PROGRAM MAIN
VAR
	Axis1 : AXIS_REF;
	
	PowerAxis1 : MC_Power;
	PowerAxis1Out : ST_McOutputs;
	
	ResetAxis1 : MC_Reset;
	ResetAxis1Out : ST_McOutputs;
	
	MoveAxis1 : MC_MoveAbsolute();
	MoveAxis2 : MC_MoveAbsolute;
	MoveAbsolute1 : ST_McOutputs;
	MoveAbsolute2 : ST_McOutputs;
	
	
	state : MoveState;
	
END_VAR


	(* update the axis status at the beginning of each cycle *)
	Axis1();
	
	(* move axis using a state machine *)
	CASE state OF
		
		MOVE_INIT :
			MoveAxis1.Execute := FALSE;
			MoveAxis2.Execute := FALSE;
			ResetAxis1.Execute := FALSE;
			state := MOVE_ENABLE;
		
		MOVE_ENABLE:
			PowerAxis1.Enable := TRUE;
			PowerAxis1.Enable_Positive := TRUE;
			PowerAxis1.Enable_Negative := TRUE;
			IF PowerAxis1.Status THEN
				state := MOVE_MOVEFORWARD;
			ELSIF PowerAxis1.Error THEN	
				state := MOVE_ERROR;
			END_IF
		MOVE_MOVEFORWARD:
			MoveAxis1.Execute := TRUE;
			MoveAxis1.Position := 500;
			MoveAxis1.Velocity := 500;
			
			IF MoveAxis1.Error THEN
				state := MOVE_ERROR;
			ELSIF MoveAxis1.Done THEN
				MoveAxis1.Execute := FALSE;
				state := MOVE_MOVEBACKWARD;
			END_IF
			
		MOVE_MOVEBACKWARD:
			MoveAxis1.Execute := TRUE;
			MoveAxis1.Position := 0;
			MoveAxis1.Velocity := 500;
			
			IF MoveAxis1.Error THEN
				state := MOVE_ERROR;
			ELSIF MoveAxis1.Done THEN
				MoveAxis1.Execute := FALSE;
				state := MOVE_MOVEFORWARD;
			END_IF
		MOVE_ERROR:
			//DO nothing here
		MOVE_RESET:
			//DO nothing here
	END_CASE
	
	ActPower();	(* call the power function block *)
	ActMove();	(* call the move function block *)
	ActReset();	(* call the reset function block *)

ACTION ActMove:
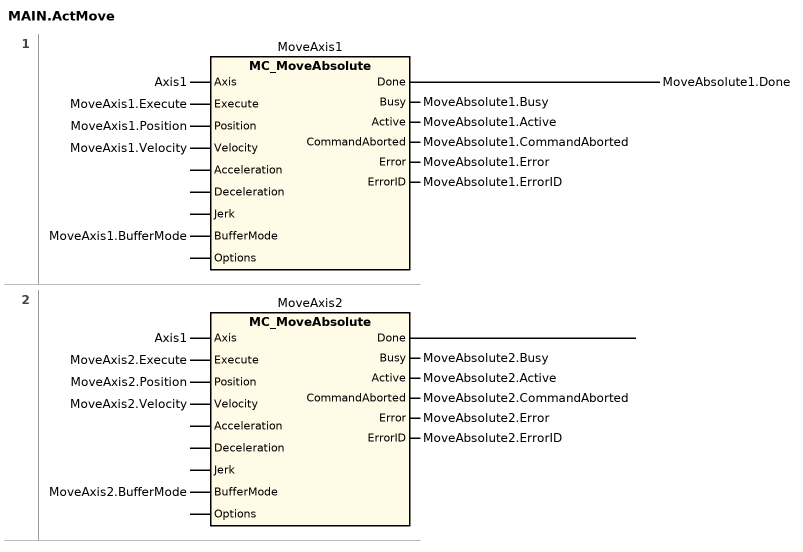
// NETWORK 1
MoveAxis1(
    Axis := Axis1,
    Execute := MoveAxis1.Execute,
    Position := MoveAxis1.Position,
    Velocity := MoveAxis1.Velocity,
    BufferMode := MoveAxis1.BufferMode,
    Busy => MoveAbsolute1.Busy,
    Active => MoveAbsolute1.Active,
    CommandAborted => MoveAbsolute1.CommandAborted,
    Error => MoveAbsolute1.Error,
    ErrorID => MoveAbsolute1.ErrorID); // MC_MoveAbsolute
MoveAbsolute1.Done := MoveAxis1.Done;

// NETWORK 2
MoveAxis2(
    Axis := Axis1,
    Execute := MoveAxis2.Execute,
    Position := MoveAxis2.Position,
    Velocity := MoveAxis2.Velocity,
    BufferMode := MoveAxis2.BufferMode,
    Busy => MoveAbsolute2.Busy,
    Active => MoveAbsolute2.Active,
    CommandAborted => MoveAbsolute2.CommandAborted,
    Error => MoveAbsolute2.Error,
    ErrorID => MoveAbsolute2.ErrorID); // MC_MoveAbsolute
END_ACTION

ACTION ActPower:
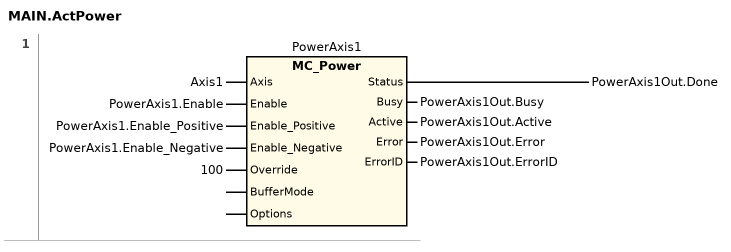
// NETWORK 1
PowerAxis1(
    Axis := Axis1,
    Enable := PowerAxis1.Enable,
    Enable_Positive := PowerAxis1.Enable_Positive,
    Enable_Negative := PowerAxis1.Enable_Negative,
    Override := 100,
    Busy => PowerAxis1Out.Busy,
    Active => PowerAxis1Out.Active,
    Error => PowerAxis1Out.Error,
    ErrorID => PowerAxis1Out.ErrorID); // MC_Power
PowerAxis1Out.Done := PowerAxis1.Status;
END_ACTION

ACTION ActReset:
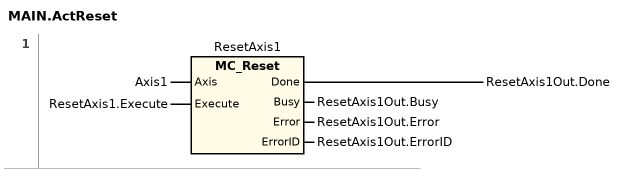
// NETWORK 1
ResetAxis1(
    Axis := Axis1,
    Execute := ResetAxis1.Execute,
    Busy => ResetAxis1Out.Busy,
    Error => ResetAxis1Out.Error,
    ErrorID => ResetAxis1Out.ErrorID); // MC_Reset
ResetAxis1Out.Done := ResetAxis1.Done;
END_ACTION

END_PROGRAM

(* stored: Version 1.1.0.1, ProductVersion 3.1.4024.12
   POU MAIN: Id {3fae0c4d-d145-4b7e-8c19-5417be10b314}, SpecialFunc None
   Action ActMove: Id {2958b60a-b494-489a-adb7-d66f216f7319}
   Action ActPower: Id {a70890ea-c1e2-4b29-9ee5-b0591beafc39}
   Action ActReset: Id {08e18cca-746f-4ca9-9e89-562807d0ba3f} *)
